// TIA Portal project "Tartak_Projekt" (V14)

(* hardware
DEVICE "S7-1200 station_1"  S7-1200 Station
   slot 0: "Rack_0"  S7-1200 Rack  Rack  V1.0
   slot 1: "PLC_1"  CPU 1214C DC/DC/DC  6ES7 214-1AG31-0XB0  V3.0
      slot 3: "AQ 1x12BIT_1"  AQ1 signal board  6ES7 232-4HA30-0XB0  V1.0
   slot 2: "DI 16/DQ 16x24VDC_1"  SM 1223 DI16/DQ16 x 24VDC  6ES7 223-1BL30-0XB0  V1.0
DEVICE "HMI_2"  TP700 Comfort
   slot 0: "TP700 Comfort"  TP700 Comfort  6AV2 124-0GC01-0AX0  14.0.1.0
   slot 1: "HMI_RT_2"  TP700 Comfort  6AV2 124-0GC01-0AX0  14.0.1.0
   slot 5: "HMI_1.IE_CP_1"  PROFINET Interface  14.0.1.0
      slot 1: "PROFINET Interface_1"  PROFINET Interface
         slot 1: "Port_1"  Port
         slot 2: "Port_2"  Port
   slot 7: "HMI_1.MPI/DP_CP_1"  MPI/DP Interface  14.0.1.0
*)

// ===== PLC "PLC_1"  CPU 1214C DC/DC/DC =====

VAR_GLOBAL   // PLC tag table "Non Default tag table2"
   "Tag_1" AT %M100.0 : Bool;
   "Tag_2" AT %M100.1 : Bool;
   "Tag_3" AT %M100.2 : Bool;
   "Tag_4" AT %M100.3 : Bool;
   "Tag_5" AT %M100.4 : Bool;
   "Tag_6" AT %M100.5 : Bool;
END_VAR

VAR_GLOBAL   // PLC tag table "Default tag table"
   "polozenie_dluga" AT %I8.0 : Bool;
   "polozenie_srednia" AT %I8.1 : Bool;
   "polozenie_krotka" AT %I8.2 : Bool;
   "polozenie_zsyp_krotki" AT %I8.3 : Bool;
   "polozenie_zsyp_sredni" AT %I8.4 : Bool;
   "polozenie_zsyp_dlugi" AT %I8.5 : Bool;
   "P1" AT %Q4.0 : Bool;   // Przepychacz belek krótkich
   "P2" AT %Q4.1 : Bool;   // Przepychacz belek średnich
   "P3" AT %Q4.2 : Bool;   // Przepychacz belek długich
   "otwarcie_zsyp_krotki" AT %Q4.3 : Bool;
   "otwarcie_zsyp_sredni" AT %Q4.4 : Bool;
   "otwarcie_zsyp_dlugi" AT %Q4.5 : Bool;
   "napelnienie_zsyp_krotki" AT %I8.6 : Bool;
   "napelnienie_zsyp_sredni" AT %I8.7 : Bool;
   "napelnienie_zsyp_dlugi" AT %I9.0 : Bool;
   "pozycja_wagnik_zsyp_krotki" AT %I9.7 : Bool;
   "pozycja_wagonik_zsyp_sredni" AT %I1.0 : Bool;
   "pozycja_wagonik_zsyp_dlugi" AT %I1.1 : Bool;
   "ruch_wagonika" AT %Q4.6 : Bool;
   "zwrotnica_bit_0" AT %Q4.7 : Bool;
   "zwrotnica_bit_1" AT %Q5.0 : Bool;
   "bocznica_krotka_0" AT %I9.1 : Bool;
   "bocznica_krotka_1" AT %I9.2 : Bool;
   "bocznica_srednia_0" AT %I9.3 : Bool;
   "bocznica_srednia_1" AT %I9.4 : Bool;
   "bocznica_dluga_0" AT %I9.5 : Bool;
   "bocznica_dluga_1" AT %I9.6 : Bool;
   "sygnalizator_dlugi" AT %Q5.1 : Bool;
   "sygnalizator_sredni" AT %Q5.2 : Bool;
   "sygnalizator_krotki" AT %Q5.3 : Bool;
   "Clock_Byte" AT %MB0 : Byte;
   "Clock_10Hz" AT %M0.0 : Bool;
   "Clock_5Hz" AT %M0.1 : Bool;
   "Clock_2.5Hz" AT %M0.2 : Bool;
   "Clock_2Hz" AT %M0.3 : Bool;
   "Clock_1.25Hz" AT %M0.4 : Bool;
   "Clock_1Hz" AT %M0.5 : Bool;
   "Clock_0.625Hz" AT %M0.6 : Bool;
   "Clock_0.5Hz" AT %M0.7 : Bool;
   "alarmy" AT %MW10 : Int;
END_VAR

VAR_GLOBAL CONSTANT   // PLC tag table "Default tag table"
   "None" : Pip := 65535;
   "Automatic update" : Pip := 0;
   "PIP 1" : Pip := 1;
   "PIP 2" : Pip := 2;
   "PIP 3" : Pip := 3;
   "PIP 4" : Pip := 4;
   "PIP OB Servo" : Pip := 32768;
   "Local~MC" : Hw_SubModule := 51;
   "Local~Common" : Hw_SubModule := 50;
   "Local~Device" : Hw_Device := 32;
   "Local~Configuration" : Hw_SubModule := 33;
   "Local~Exec" : Hw_SubModule := 52;
   "Local(1)" : Hw_SubModule := 49;
   "Local~PROFINET_interface_1(1)" : Hw_Interface := 64;
   "Local~PROFINET_interface_1~Port_1(1)" : Hw_Interface := 65;
   "Local~HSC_1(1)" : Hw_Hsc := 257;
   "Local~HSC_2(1)" : Hw_Hsc := 258;
   "Local~HSC_3(1)" : Hw_Hsc := 259;
   "Local~HSC_4(1)" : Hw_Hsc := 260;
   "Local~HSC_5(1)" : Hw_Hsc := 261;
   "Local~HSC_6(1)" : Hw_Hsc := 262;
   "Local~AI_2_1(1)" : Hw_SubModule := 263;
   "Local~DI_14_DQ_10_1(1)" : Hw_SubModule := 264;
   "Local~Pulse_1(1)" : Hw_Pwm := 265;
   "Local~Pulse_2(1)" : Hw_Pwm := 266;
   "Local~Pulse_3(1)" : Hw_Pwm := 267;
   "Local~Pulse_4(1)" : Hw_Pwm := 268;
   "OB_Main(1)" : OB_PCYCLE := 1;
END_VAR

DATA_BLOCK "DB_HMI"   // DB1
{ S7_Optimized_Access := 'TRUE' }
VERSION : 0.1
   VAR
      napelnienie_zsyp_krotki : Bool;
      napelnienie_zsyp_sredni : Bool;
      napelnienie_zsyp_dlugi : Bool;
      belka_krotka : Bool;
      belka_srednia : Bool;
      belka_dluga : Bool;
      status_ruchu_wagonika : Bool;
      oproznianie_zsyp_krotki : Bool;
      oproznianie_zsyp_sredni : Bool;
      oproznianie_zsyp_dlugi : Bool;
      ustawienie_zwrotnicy : Byte;
      zapelnienie_bocznicy_krotkiej : Byte;
      zapelnienie_bocznicy_sredniej : Byte;
      zapelnienie_bocznicy_dlugiej : Byte;
      sygnalizator_bocznica_krotka : Bool;
      sygnalizator_bocznica_srednia : Bool;
      sygnalizator_bocznica_dluga : Bool;
      wagonik_krotki : Bool;
      wagonik_sredni : Bool;
      wagonik_dlugi : Bool;
   END_VAR
BEGIN
END_DATA_BLOCK

DATA_BLOCK "wykrywanie_belki_i_zrzuczanie_DB"   // DB2
{ S7_Optimized_Access := 'TRUE' }
VERSION : 0.1
// stored: InstanceOfName wykrywanie_belki_i_zrzuczanie
"wykrywanie_belki_i_zrzuczanie"
BEGIN
END_DATA_BLOCK

DATA_BLOCK "poruszanie_wagonikiem_i_zsypywaanie_drewna_2_DB"   // DB3
{ S7_Optimized_Access := 'TRUE' }
VERSION : 0.1
// stored: InstanceOfName poruszanie_wagonikiem_i_zsypywaanie_drewna_2
"poruszanie_wagonikiem_i_zsypywaanie_drewna_2"
BEGIN
END_DATA_BLOCK

// folder: System blocks/Program resources

DATA_BLOCK "IEC_Timer_0_DB"   // DB4
{ S7_Optimized_Access := 'TRUE' }
AUTHOR : Simatic
FAMILY : IEC
NAME : IEC_TMR
VERSION : 1.0
// stored: InstanceOfName IEC_TIMER
"IEC_TIMER"
BEGIN
END_DATA_BLOCK

// folder: (top level)

FUNCTION_BLOCK "wykrywanie_belki_i_zrzuczanie"   // FB1, LAD
{ S7_Optimized_Access := 'TRUE' }
VERSION : 0.1
   VAR
      czy_wykryta_belka : Bool;
      krotka_belka : Bool;
      srednia_belka : Bool;
      dluga_belka : Bool;
      belka_zrzucona : Bool;
   END_VAR
   VAR_TEMP
      belka_na_pomiarze : Bool;
   END_VAR
   VAR_TEMP   // added for the SCL form of the ladder/FBD networks
      _w1 : Bool;
      _w2 : Bool;
      _w3 : Bool;
      _w4 : Bool;
   END_VAR
BEGIN

REGION Network 1
   // Czy belka jest już na pomiarze?
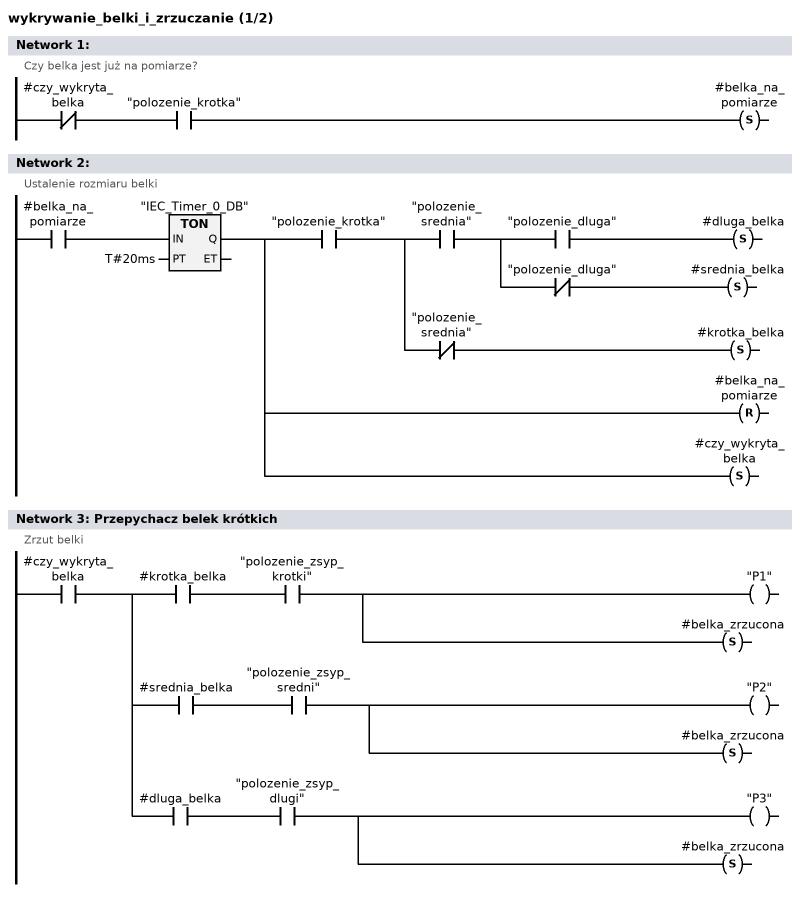
   RUNG wire#powerrail
      I_Contact( #czy_wykryta_belka )
      Contact( "polozenie_krotka" )
      S_Coil( #belka_na_pomiarze )
   END_RUNG
   // the same network as SCL:
   IF NOT #czy_wykryta_belka AND "polozenie_krotka" THEN #belka_na_pomiarze := TRUE; END_IF;
END_REGION

REGION Network 2
   // Ustalenie rozmiaru belki
   "IEC_Timer_0_DB".TON(IN := #belka_na_pomiarze, PT := T#20ms);
   #_w1 := "IEC_Timer_0_DB".Q AND "polozenie_krotka";
   #_w2 := #_w1 AND "polozenie_srednia";
   IF #_w2 AND "polozenie_dluga" THEN #dluga_belka := TRUE; END_IF;
   IF #_w2 AND NOT "polozenie_dluga" THEN #srednia_belka := TRUE; END_IF;
   IF #_w1 AND NOT "polozenie_srednia" THEN #krotka_belka := TRUE; END_IF;
   IF "IEC_Timer_0_DB".Q THEN
       #belka_na_pomiarze := FALSE;
       #czy_wykryta_belka := TRUE;
   END_IF;
END_REGION

REGION Network 3: Przepychacz belek krótkich
   // Zrzut belki
   RUNG wire#powerrail
      Contact( #czy_wykryta_belka )
      wire#w1
      Contact( #krotka_belka )
      Contact( "polozenie_zsyp_krotki" )
      wire#w2
      Coil( "P1" )
   END_RUNG
   RUNG wire#w2
      S_Coil( #belka_zrzucona )
   END_RUNG
   RUNG wire#w1
      Contact( #srednia_belka )
      Contact( "polozenie_zsyp_sredni" )
      wire#w3
      Coil( "P2" )
   END_RUNG
   RUNG wire#w3
      S_Coil( #belka_zrzucona )
   END_RUNG
   RUNG wire#w1
      Contact( #dluga_belka )
      Contact( "polozenie_zsyp_dlugi" )
      wire#w4
      Coil( "P3" )
   END_RUNG
   RUNG wire#w4
      S_Coil( #belka_zrzucona )
   END_RUNG
   // the same network as SCL:
   "P1" := #czy_wykryta_belka AND #krotka_belka AND "polozenie_zsyp_krotki";
   IF "P1" THEN #belka_zrzucona := TRUE; END_IF;
   "P2" := #czy_wykryta_belka AND #srednia_belka AND "polozenie_zsyp_sredni";
   IF "P2" THEN #belka_zrzucona := TRUE; END_IF;
   "P3" := #czy_wykryta_belka AND #dluga_belka AND "polozenie_zsyp_dlugi";
   IF "P3" THEN #belka_zrzucona := TRUE; END_IF;
END_REGION

REGION Network 4: Przepychacz belek krótkich
   // Czekamy, aż belka zostanie zrzucona
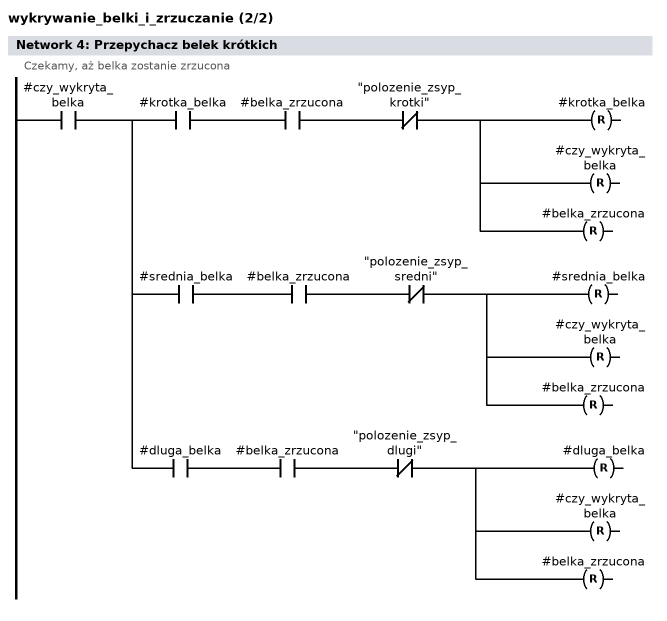
   RUNG wire#powerrail
      Contact( #czy_wykryta_belka )
      wire#w1
      Contact( #krotka_belka )
      Contact( #belka_zrzucona )
      I_Contact( "polozenie_zsyp_krotki" )
      wire#w2
      R_Coil( #krotka_belka )
   END_RUNG
   RUNG wire#w2
      R_Coil( #czy_wykryta_belka )
   END_RUNG
   RUNG wire#w2
      R_Coil( #belka_zrzucona )
   END_RUNG
   RUNG wire#w1
      Contact( #srednia_belka )
      Contact( #belka_zrzucona )
      I_Contact( "polozenie_zsyp_sredni" )
      wire#w3
      R_Coil( #srednia_belka )
   END_RUNG
   RUNG wire#w3
      R_Coil( #czy_wykryta_belka )
   END_RUNG
   RUNG wire#w3
      R_Coil( #belka_zrzucona )
   END_RUNG
   RUNG wire#w1
      Contact( #dluga_belka )
      Contact( #belka_zrzucona )
      I_Contact( "polozenie_zsyp_dlugi" )
      wire#w4
      R_Coil( #dluga_belka )
   END_RUNG
   RUNG wire#w4
      R_Coil( #czy_wykryta_belka )
   END_RUNG
   RUNG wire#w4
      R_Coil( #belka_zrzucona )
   END_RUNG
   // the same network as SCL:
   #_w1 := #czy_wykryta_belka AND #krotka_belka AND #belka_zrzucona AND NOT "polozenie_zsyp_krotki";
   IF #_w1 THEN #krotka_belka := FALSE; END_IF;
   #_w2 := #czy_wykryta_belka;
   IF #_w1 THEN
       #czy_wykryta_belka := FALSE;
       #belka_zrzucona := FALSE;
   END_IF;
   #_w3 := #_w2 AND #srednia_belka AND #belka_zrzucona AND NOT "polozenie_zsyp_sredni";
   IF #_w3 THEN
       #srednia_belka := FALSE;
       #czy_wykryta_belka := FALSE;
       #belka_zrzucona := FALSE;
   END_IF;
   #_w4 := #_w2 AND #dluga_belka AND #belka_zrzucona AND NOT "polozenie_zsyp_dlugi";
   IF #_w4 THEN
       #dluga_belka := FALSE;
       #czy_wykryta_belka := FALSE;
       #belka_zrzucona := FALSE;
   END_IF;
END_REGION
END_FUNCTION_BLOCK

FUNCTION_BLOCK "poruszanie_wagonikiem_i_zsypywaanie_drewna_2"   // FB2, LAD
{ S7_Optimized_Access := 'TRUE' }
VERSION : 0.1
   VAR
      wagonik_krotki : Bool;
      wagonik_sredni : Bool;
      wagonik_dlugi : Bool;
   END_VAR
   VAR_TEMP   // added for the SCL form of the ladder/FBD networks
      _w1 : Bool;
      _w2 : Bool;
      _w3 : Bool;
      _w4 : Bool;
      _w5 : Bool;
      _w6 : Bool;
   END_VAR
BEGIN

REGION Network 1
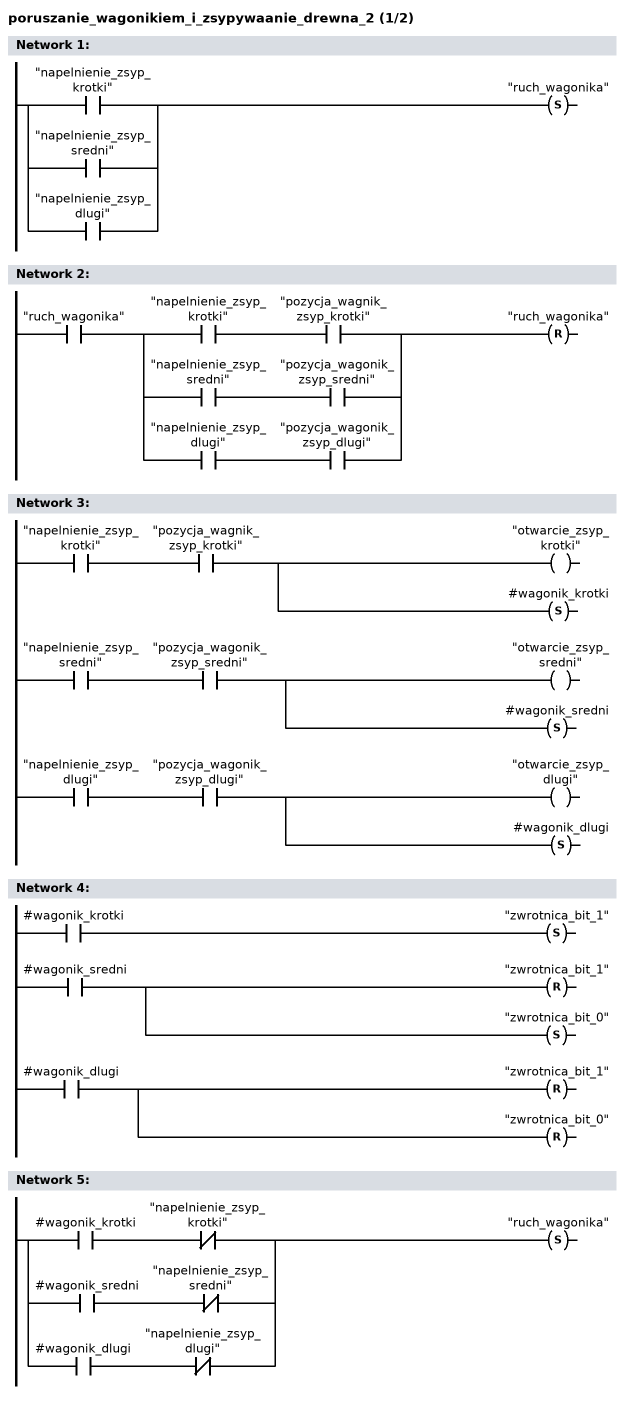
   RUNG wire#powerrail
      Contact( "napelnienie_zsyp_krotki" )
      wire#w1
      S_Coil( "ruch_wagonika" )
   END_RUNG
   RUNG wire#powerrail
      Contact( "napelnienie_zsyp_sredni" )
   END_RUNG wire#w1
   RUNG wire#powerrail
      Contact( "napelnienie_zsyp_dlugi" )
   END_RUNG wire#w1
   // the same network as SCL:
   IF "napelnienie_zsyp_krotki" OR "napelnienie_zsyp_sredni" OR "napelnienie_zsyp_dlugi" THEN
       "ruch_wagonika" := TRUE;
   END_IF;
END_REGION

REGION Network 2
   RUNG wire#powerrail
      Contact( "ruch_wagonika" )
      wire#w1
      Contact( "napelnienie_zsyp_krotki" )
      Contact( "pozycja_wagnik_zsyp_krotki" )
      wire#w2
      R_Coil( "ruch_wagonika" )
   END_RUNG
   RUNG wire#w1
      Contact( "napelnienie_zsyp_sredni" )
      Contact( "pozycja_wagonik_zsyp_sredni" )
   END_RUNG wire#w2
   RUNG wire#w1
      Contact( "napelnienie_zsyp_dlugi" )
      Contact( "pozycja_wagonik_zsyp_dlugi" )
   END_RUNG wire#w2
   // the same network as SCL:
   IF "ruch_wagonika" AND (("napelnienie_zsyp_krotki" AND "pozycja_wagnik_zsyp_krotki") OR ("napelnienie_zsyp_sredni" AND "pozycja_wagonik_zsyp_sredni") OR ("napelnienie_zsyp_dlugi" AND "pozycja_wagonik_zsyp_dlugi")) THEN
       "ruch_wagonika" := FALSE;
   END_IF;
END_REGION

REGION Network 3
   RUNG wire#powerrail
      Contact( "napelnienie_zsyp_krotki" )
      Contact( "pozycja_wagnik_zsyp_krotki" )
      wire#w1
      Coil( "otwarcie_zsyp_krotki" )
   END_RUNG
   RUNG wire#w1
      S_Coil( #wagonik_krotki )
   END_RUNG
   RUNG wire#powerrail
      Contact( "napelnienie_zsyp_sredni" )
      Contact( "pozycja_wagonik_zsyp_sredni" )
      wire#w2
      Coil( "otwarcie_zsyp_sredni" )
   END_RUNG
   RUNG wire#w2
      S_Coil( #wagonik_sredni )
   END_RUNG
   RUNG wire#powerrail
      Contact( "napelnienie_zsyp_dlugi" )
      Contact( "pozycja_wagonik_zsyp_dlugi" )
      wire#w3
      Coil( "otwarcie_zsyp_dlugi" )
   END_RUNG
   RUNG wire#w3
      S_Coil( #wagonik_dlugi )
   END_RUNG
   // the same network as SCL:
   "otwarcie_zsyp_krotki" := "napelnienie_zsyp_krotki" AND "pozycja_wagnik_zsyp_krotki";
   IF "otwarcie_zsyp_krotki" THEN #wagonik_krotki := TRUE; END_IF;
   "otwarcie_zsyp_sredni" := "napelnienie_zsyp_sredni" AND "pozycja_wagonik_zsyp_sredni";
   IF "otwarcie_zsyp_sredni" THEN #wagonik_sredni := TRUE; END_IF;
   "otwarcie_zsyp_dlugi" := "napelnienie_zsyp_dlugi" AND "pozycja_wagonik_zsyp_dlugi";
   IF "otwarcie_zsyp_dlugi" THEN #wagonik_dlugi := TRUE; END_IF;
END_REGION

REGION Network 4
   RUNG wire#powerrail
      Contact( #wagonik_krotki )
      S_Coil( "zwrotnica_bit_1" )
   END_RUNG
   RUNG wire#powerrail
      Contact( #wagonik_sredni )
      wire#w1
      R_Coil( "zwrotnica_bit_1" )
   END_RUNG
   RUNG wire#w1
      S_Coil( "zwrotnica_bit_0" )
   END_RUNG
   RUNG wire#powerrail
      Contact( #wagonik_dlugi )
      wire#w2
      R_Coil( "zwrotnica_bit_1" )
   END_RUNG
   RUNG wire#w2
      R_Coil( "zwrotnica_bit_0" )
   END_RUNG
   // the same network as SCL:
   IF #wagonik_krotki THEN "zwrotnica_bit_1" := TRUE; END_IF;
   IF #wagonik_sredni THEN
       "zwrotnica_bit_1" := FALSE;
       "zwrotnica_bit_0" := TRUE;
   END_IF;
   IF #wagonik_dlugi THEN
       "zwrotnica_bit_1" := FALSE;
       "zwrotnica_bit_0" := FALSE;
   END_IF;
END_REGION

REGION Network 5
   RUNG wire#powerrail
      Contact( #wagonik_krotki )
      I_Contact( "napelnienie_zsyp_krotki" )
      wire#w1
      S_Coil( "ruch_wagonika" )
   END_RUNG
   RUNG wire#powerrail
      Contact( #wagonik_sredni )
      I_Contact( "napelnienie_zsyp_sredni" )
   END_RUNG wire#w1
   RUNG wire#powerrail
      Contact( #wagonik_dlugi )
      I_Contact( "napelnienie_zsyp_dlugi" )
   END_RUNG wire#w1
   // the same network as SCL:
   IF (#wagonik_krotki AND NOT "napelnienie_zsyp_krotki") OR (#wagonik_sredni AND NOT "napelnienie_zsyp_sredni") OR (#wagonik_dlugi AND NOT "napelnienie_zsyp_dlugi") THEN
       "ruch_wagonika" := TRUE;
   END_IF;
END_REGION

REGION Network 6
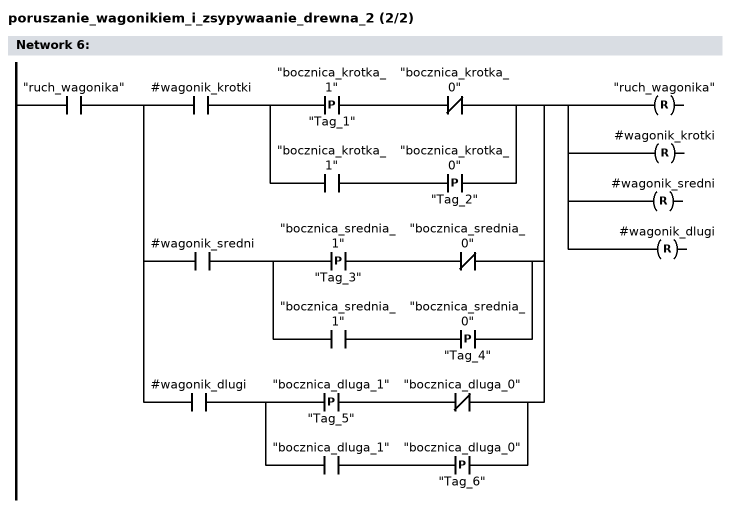
   RUNG wire#powerrail
      Contact( "ruch_wagonika" )
      wire#w1
      Contact( #wagonik_krotki )
      wire#w2
      P_Contact(operand := "bocznica_krotka_1", bit := "Tag_1")
      I_Contact( "bocznica_krotka_0" )
      wire#w3
      R_Coil( "ruch_wagonika" )
   END_RUNG
   RUNG wire#w2
      Contact( "bocznica_krotka_1" )
      P_Contact(operand := "bocznica_krotka_0", bit := "Tag_2")
   END_RUNG wire#w3
   RUNG wire#w1
      Contact( #wagonik_sredni )
      wire#w4
      P_Contact(operand := "bocznica_srednia_1", bit := "Tag_3")
      I_Contact( "bocznica_srednia_0" )
   END_RUNG wire#w3
   RUNG wire#w4
      Contact( "bocznica_srednia_1" )
      P_Contact(operand := "bocznica_srednia_0", bit := "Tag_4")
   END_RUNG wire#w3
   RUNG wire#w1
      Contact( #wagonik_dlugi )
      wire#w5
      P_Contact(operand := "bocznica_dluga_1", bit := "Tag_5")
      I_Contact( "bocznica_dluga_0" )
   END_RUNG wire#w3
   RUNG wire#w5
      Contact( "bocznica_dluga_1" )
      P_Contact(operand := "bocznica_dluga_0", bit := "Tag_6")
   END_RUNG wire#w3
   RUNG wire#w3
      R_Coil( #wagonik_krotki )
   END_RUNG
   RUNG wire#w3
      R_Coil( #wagonik_sredni )
   END_RUNG
   RUNG wire#w3
      R_Coil( #wagonik_dlugi )
   END_RUNG
   // the same network as SCL:
   #_w1 := "ruch_wagonika" AND #wagonik_krotki AND "bocznica_krotka_1" AND NOT "Tag_1";   // rising edge of "bocznica_krotka_1"
   "Tag_1" := "bocznica_krotka_1";
   #_w2 := "ruch_wagonika" AND #wagonik_krotki AND "bocznica_krotka_1" AND "bocznica_krotka_0" AND NOT "Tag_2";   // rising edge of "bocznica_krotka_0"
   "Tag_2" := "bocznica_krotka_0";
   #_w3 := "ruch_wagonika" AND #wagonik_sredni AND "bocznica_srednia_1" AND NOT "Tag_3";   // rising edge of "bocznica_srednia_1"
   "Tag_3" := "bocznica_srednia_1";
   #_w4 := "ruch_wagonika" AND #wagonik_sredni AND "bocznica_srednia_1" AND "bocznica_srednia_0" AND NOT "Tag_4";   // rising edge of "bocznica_srednia_0"
   "Tag_4" := "bocznica_srednia_0";
   #_w5 := "ruch_wagonika" AND #wagonik_dlugi AND "bocznica_dluga_1" AND NOT "Tag_5";   // rising edge of "bocznica_dluga_1"
   "Tag_5" := "bocznica_dluga_1";
   #_w6 := "ruch_wagonika" AND #wagonik_dlugi AND "bocznica_dluga_1" AND "bocznica_dluga_0" AND NOT "Tag_6";   // rising edge of "bocznica_dluga_0"
   "Tag_6" := "bocznica_dluga_0";
   IF (#_w1 AND NOT "bocznica_krotka_0") OR #_w2 OR (#_w3 AND NOT "bocznica_srednia_0") OR #_w4 OR (#_w5 AND NOT "bocznica_dluga_0") OR #_w6 THEN
       "ruch_wagonika" := FALSE;
       #wagonik_krotki := FALSE;
       #wagonik_sredni := FALSE;
       #wagonik_dlugi := FALSE;
   END_IF;
END_REGION
END_FUNCTION_BLOCK

FUNCTION "przepisywanie_HMI" : Void   // FC1, LAD
{ S7_Optimized_Access := 'TRUE' }
VERSION : 0.1
BEGIN

REGION Network 1: Napełnianie zsypów
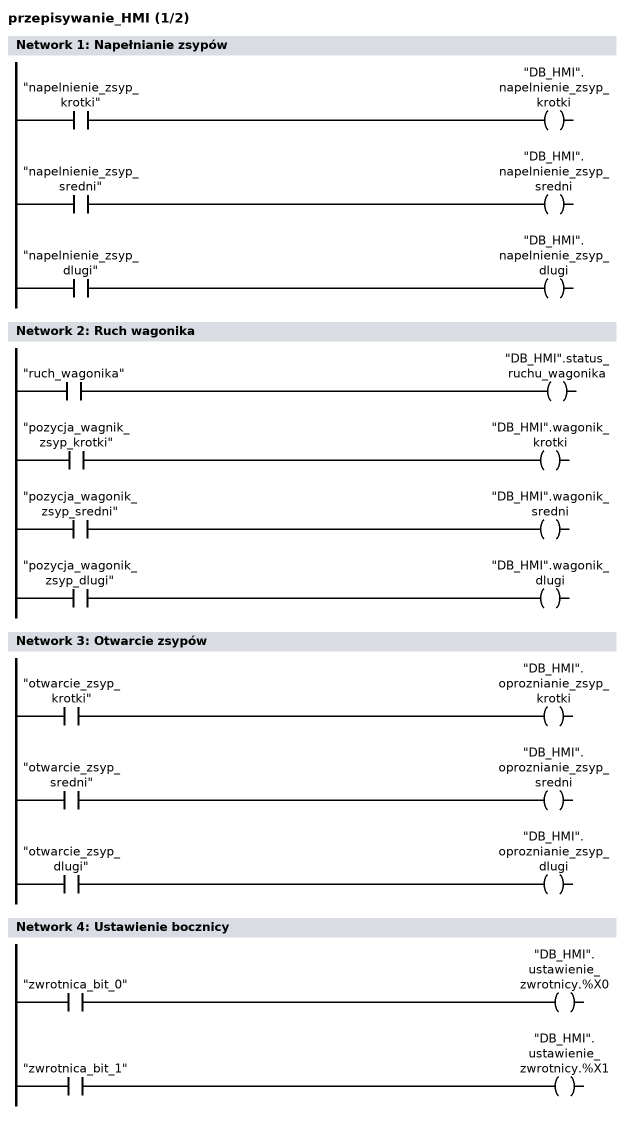
   RUNG wire#powerrail
      Contact( "napelnienie_zsyp_krotki" )
      Coil( "DB_HMI".napelnienie_zsyp_krotki )
   END_RUNG
   RUNG wire#powerrail
      Contact( "napelnienie_zsyp_sredni" )
      Coil( "DB_HMI".napelnienie_zsyp_sredni )
   END_RUNG
   RUNG wire#powerrail
      Contact( "napelnienie_zsyp_dlugi" )
      Coil( "DB_HMI".napelnienie_zsyp_dlugi )
   END_RUNG
   // the same network as SCL:
   "DB_HMI".napelnienie_zsyp_krotki := "napelnienie_zsyp_krotki";
   "DB_HMI".napelnienie_zsyp_sredni := "napelnienie_zsyp_sredni";
   "DB_HMI".napelnienie_zsyp_dlugi := "napelnienie_zsyp_dlugi";
END_REGION

REGION Network 2: Ruch wagonika
   RUNG wire#powerrail
      Contact( "ruch_wagonika" )
      Coil( "DB_HMI".status_ruchu_wagonika )
   END_RUNG
   RUNG wire#powerrail
      Contact( "pozycja_wagnik_zsyp_krotki" )
      Coil( "DB_HMI".wagonik_krotki )
   END_RUNG
   RUNG wire#powerrail
      Contact( "pozycja_wagonik_zsyp_sredni" )
      Coil( "DB_HMI".wagonik_sredni )
   END_RUNG
   RUNG wire#powerrail
      Contact( "pozycja_wagonik_zsyp_dlugi" )
      Coil( "DB_HMI".wagonik_dlugi )
   END_RUNG
   // the same network as SCL:
   "DB_HMI".status_ruchu_wagonika := "ruch_wagonika";
   "DB_HMI".wagonik_krotki := "pozycja_wagnik_zsyp_krotki";
   "DB_HMI".wagonik_sredni := "pozycja_wagonik_zsyp_sredni";
   "DB_HMI".wagonik_dlugi := "pozycja_wagonik_zsyp_dlugi";
END_REGION

REGION Network 3: Otwarcie zsypów
   RUNG wire#powerrail
      Contact( "otwarcie_zsyp_krotki" )
      Coil( "DB_HMI".oproznianie_zsyp_krotki )
   END_RUNG
   RUNG wire#powerrail
      Contact( "otwarcie_zsyp_sredni" )
      Coil( "DB_HMI".oproznianie_zsyp_sredni )
   END_RUNG
   RUNG wire#powerrail
      Contact( "otwarcie_zsyp_dlugi" )
      Coil( "DB_HMI".oproznianie_zsyp_dlugi )
   END_RUNG
   // the same network as SCL:
   "DB_HMI".oproznianie_zsyp_krotki := "otwarcie_zsyp_krotki";
   "DB_HMI".oproznianie_zsyp_sredni := "otwarcie_zsyp_sredni";
   "DB_HMI".oproznianie_zsyp_dlugi := "otwarcie_zsyp_dlugi";
END_REGION

REGION Network 4: Ustawienie bocznicy
   RUNG wire#powerrail
      Contact( "zwrotnica_bit_0" )
      Coil( "DB_HMI".ustawienie_zwrotnicy.%X0 )
   END_RUNG
   RUNG wire#powerrail
      Contact( "zwrotnica_bit_1" )
      Coil( "DB_HMI".ustawienie_zwrotnicy.%X1 )
   END_RUNG
   // the same network as SCL:
   "DB_HMI".ustawienie_zwrotnicy.%X0 := "zwrotnica_bit_0";
   "DB_HMI".ustawienie_zwrotnicy.%X1 := "zwrotnica_bit_1";
END_REGION

REGION Network 5: Zapełnienie bocznic
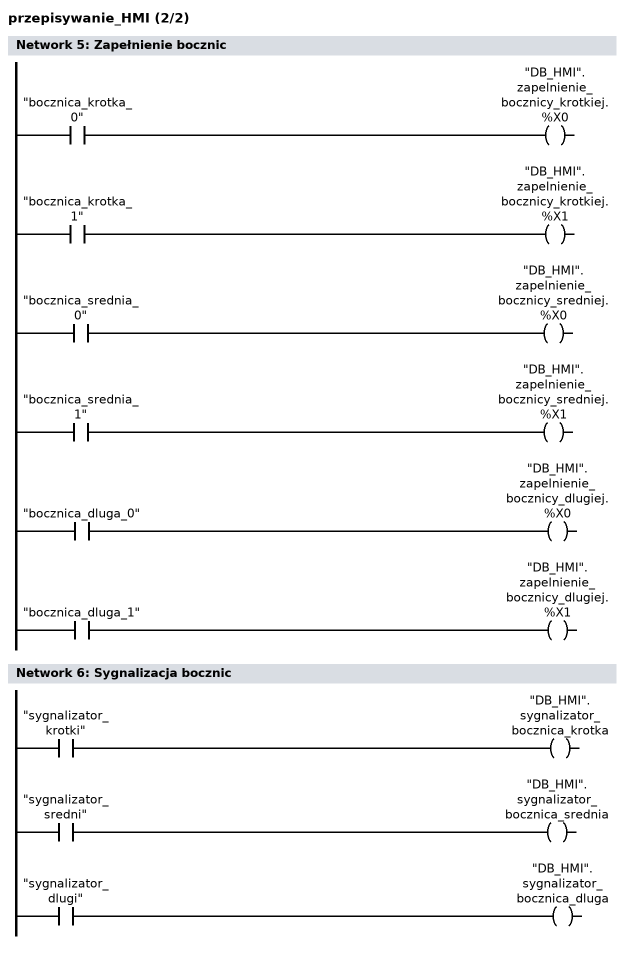
   RUNG wire#powerrail
      Contact( "bocznica_krotka_0" )
      Coil( "DB_HMI".zapelnienie_bocznicy_krotkiej.%X0 )
   END_RUNG
   RUNG wire#powerrail
      Contact( "bocznica_krotka_1" )
      Coil( "DB_HMI".zapelnienie_bocznicy_krotkiej.%X1 )
   END_RUNG
   RUNG wire#powerrail
      Contact( "bocznica_srednia_0" )
      Coil( "DB_HMI".zapelnienie_bocznicy_sredniej.%X0 )
   END_RUNG
   RUNG wire#powerrail
      Contact( "bocznica_srednia_1" )
      Coil( "DB_HMI".zapelnienie_bocznicy_sredniej.%X1 )
   END_RUNG
   RUNG wire#powerrail
      Contact( "bocznica_dluga_0" )
      Coil( "DB_HMI".zapelnienie_bocznicy_dlugiej.%X0 )
   END_RUNG
   RUNG wire#powerrail
      Contact( "bocznica_dluga_1" )
      Coil( "DB_HMI".zapelnienie_bocznicy_dlugiej.%X1 )
   END_RUNG
   // the same network as SCL:
   "DB_HMI".zapelnienie_bocznicy_krotkiej.%X0 := "bocznica_krotka_0";
   "DB_HMI".zapelnienie_bocznicy_krotkiej.%X1 := "bocznica_krotka_1";
   "DB_HMI".zapelnienie_bocznicy_sredniej.%X0 := "bocznica_srednia_0";
   "DB_HMI".zapelnienie_bocznicy_sredniej.%X1 := "bocznica_srednia_1";
   "DB_HMI".zapelnienie_bocznicy_dlugiej.%X0 := "bocznica_dluga_0";
   "DB_HMI".zapelnienie_bocznicy_dlugiej.%X1 := "bocznica_dluga_1";
END_REGION

REGION Network 6: Sygnalizacja bocznic
   RUNG wire#powerrail
      Contact( "sygnalizator_krotki" )
      Coil( "DB_HMI".sygnalizator_bocznica_krotka )
   END_RUNG
   RUNG wire#powerrail
      Contact( "sygnalizator_sredni" )
      Coil( "DB_HMI".sygnalizator_bocznica_srednia )
   END_RUNG
   RUNG wire#powerrail
      Contact( "sygnalizator_dlugi" )
      Coil( "DB_HMI".sygnalizator_bocznica_dluga )
   END_RUNG
   // the same network as SCL:
   "DB_HMI".sygnalizator_bocznica_krotka := "sygnalizator_krotki";
   "DB_HMI".sygnalizator_bocznica_srednia := "sygnalizator_sredni";
   "DB_HMI".sygnalizator_bocznica_dluga := "sygnalizator_dlugi";
END_REGION
END_FUNCTION

FUNCTION "poruszanie_wagonikiem_i_zsypywanie_drewna" : Void   // FC2, LAD
{ S7_Optimized_Access := 'TRUE' }
VERSION : 0.1
BEGIN

REGION Network 1
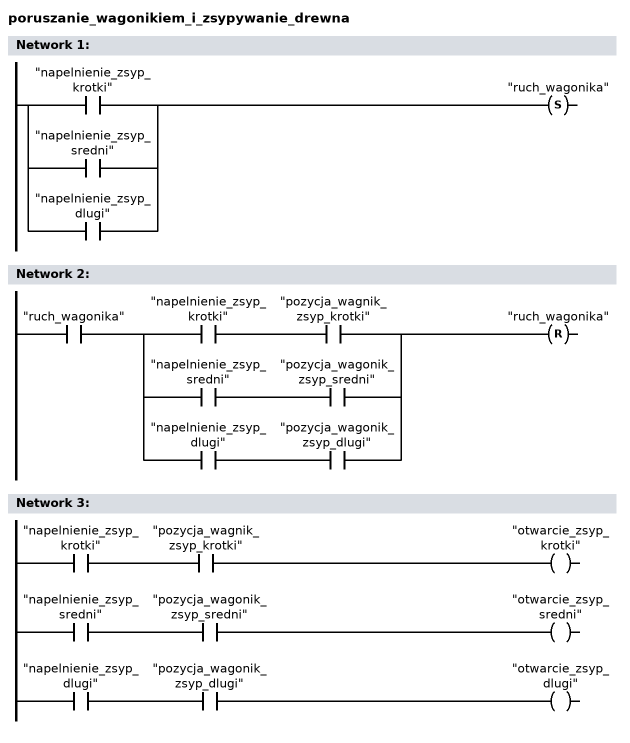
   RUNG wire#powerrail
      Contact( "napelnienie_zsyp_krotki" )
      wire#w1
      S_Coil( "ruch_wagonika" )
   END_RUNG
   RUNG wire#powerrail
      Contact( "napelnienie_zsyp_sredni" )
   END_RUNG wire#w1
   RUNG wire#powerrail
      Contact( "napelnienie_zsyp_dlugi" )
   END_RUNG wire#w1
   // the same network as SCL:
   IF "napelnienie_zsyp_krotki" OR "napelnienie_zsyp_sredni" OR "napelnienie_zsyp_dlugi" THEN
       "ruch_wagonika" := TRUE;
   END_IF;
END_REGION

REGION Network 2
   RUNG wire#powerrail
      Contact( "ruch_wagonika" )
      wire#w1
      Contact( "napelnienie_zsyp_krotki" )
      Contact( "pozycja_wagnik_zsyp_krotki" )
      wire#w2
      R_Coil( "ruch_wagonika" )
   END_RUNG
   RUNG wire#w1
      Contact( "napelnienie_zsyp_sredni" )
      Contact( "pozycja_wagonik_zsyp_sredni" )
   END_RUNG wire#w2
   RUNG wire#w1
      Contact( "napelnienie_zsyp_dlugi" )
      Contact( "pozycja_wagonik_zsyp_dlugi" )
   END_RUNG wire#w2
   // the same network as SCL:
   IF "ruch_wagonika" AND (("napelnienie_zsyp_krotki" AND "pozycja_wagnik_zsyp_krotki") OR ("napelnienie_zsyp_sredni" AND "pozycja_wagonik_zsyp_sredni") OR ("napelnienie_zsyp_dlugi" AND "pozycja_wagonik_zsyp_dlugi")) THEN
       "ruch_wagonika" := FALSE;
   END_IF;
END_REGION

REGION Network 3
   RUNG wire#powerrail
      Contact( "napelnienie_zsyp_krotki" )
      Contact( "pozycja_wagnik_zsyp_krotki" )
      Coil( "otwarcie_zsyp_krotki" )
   END_RUNG
   RUNG wire#powerrail
      Contact( "napelnienie_zsyp_sredni" )
      Contact( "pozycja_wagonik_zsyp_sredni" )
      Coil( "otwarcie_zsyp_sredni" )
   END_RUNG
   RUNG wire#powerrail
      Contact( "napelnienie_zsyp_dlugi" )
      Contact( "pozycja_wagonik_zsyp_dlugi" )
      Coil( "otwarcie_zsyp_dlugi" )
   END_RUNG
   // the same network as SCL:
   "otwarcie_zsyp_krotki" := "napelnienie_zsyp_krotki" AND "pozycja_wagnik_zsyp_krotki";
   "otwarcie_zsyp_sredni" := "napelnienie_zsyp_sredni" AND "pozycja_wagonik_zsyp_sredni";
   "otwarcie_zsyp_dlugi" := "napelnienie_zsyp_dlugi" AND "pozycja_wagonik_zsyp_dlugi";
END_REGION
END_FUNCTION

FUNCTION "opuszczanie_tartaku" : Void   // FC3, LAD
{ S7_Optimized_Access := 'TRUE' }
VERSION : 0.1
BEGIN

REGION Network 1
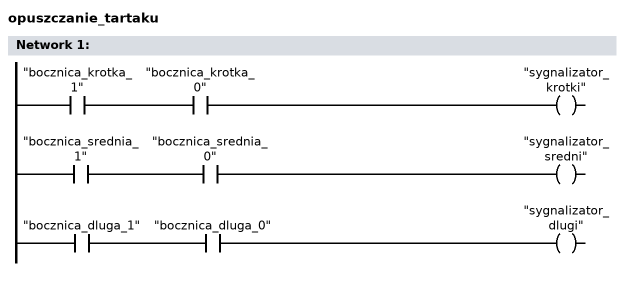
   RUNG wire#powerrail
      Contact( "bocznica_krotka_1" )
      Contact( "bocznica_krotka_0" )
      Coil( "sygnalizator_krotki" )
   END_RUNG
   RUNG wire#powerrail
      Contact( "bocznica_srednia_1" )
      Contact( "bocznica_srednia_0" )
      Coil( "sygnalizator_sredni" )
   END_RUNG
   RUNG wire#powerrail
      Contact( "bocznica_dluga_1" )
      Contact( "bocznica_dluga_0" )
      Coil( "sygnalizator_dlugi" )
   END_RUNG
   // the same network as SCL:
   "sygnalizator_krotki" := "bocznica_krotka_1" AND "bocznica_krotka_0";
   "sygnalizator_sredni" := "bocznica_srednia_1" AND "bocznica_srednia_0";
   "sygnalizator_dlugi" := "bocznica_dluga_1" AND "bocznica_dluga_0";
END_REGION
END_FUNCTION

ORGANIZATION_BLOCK "Main"   // OB1, LAD, ProgramCycle
TITLE = "Main Program Sweep (Cycle)"
{ S7_Optimized_Access := 'TRUE' }
VERSION : 0.1
   VAR_INPUT
      Initial_Call : Bool;   // Initial call of this OB
      Remanence : Bool;   // =True, if remanent data are available
   END_VAR
BEGIN

REGION Network 1
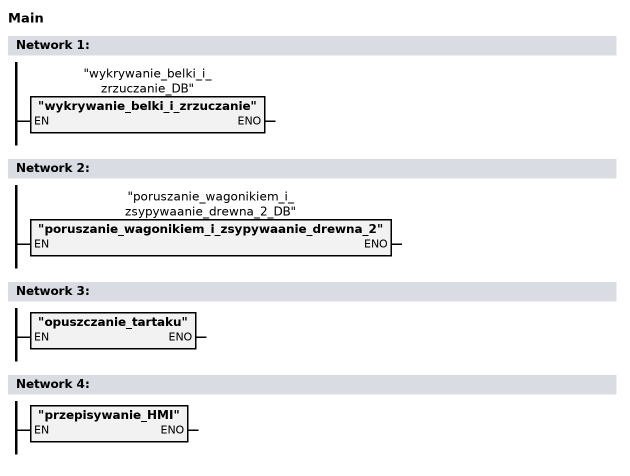
   RUNG wire#powerrail
      "wykrywanie_belki_i_zrzuczanie_DB"()
   END_RUNG
   // the same network as SCL:
   "wykrywanie_belki_i_zrzuczanie_DB"();   // "wykrywanie_belki_i_zrzuczanie"
END_REGION

REGION Network 2
   RUNG wire#powerrail
      "poruszanie_wagonikiem_i_zsypywaanie_drewna_2_DB"()
   END_RUNG
   // the same network as SCL:
   "poruszanie_wagonikiem_i_zsypywaanie_drewna_2_DB"();   // "poruszanie_wagonikiem_i_zsypywaanie_drewna_2"
END_REGION

REGION Network 3
   RUNG wire#powerrail
      "opuszczanie_tartaku"()
   END_RUNG
   // the same network as SCL:
   "opuszczanie_tartaku"();
END_REGION

REGION Network 4
   RUNG wire#powerrail
      "przepisywanie_HMI"()
   END_RUNG
   // the same network as SCL:
   "przepisywanie_HMI"();
END_REGION
END_ORGANIZATION_BLOCK

(* ===== HMI "HMI_RT_2" =====
system functions are stored by id; their names below are inferred from use
connection "HMI_Connection_1": ETHERNET, S7_1200_OMS

HMI tags "Default tag table"
   "Tag_ScreenNumber" : UInt, internal
   "DB_HMI_napelnienie_zsyp_krotki" : Bool = PLC DB_HMI.napelnienie_zsyp_krotki, 1 s
   "DB_HMI_napelnienie_zsyp_sredni" : Bool = PLC DB_HMI.napelnienie_zsyp_sredni, 1 s
   "DB_HMI_napelnienie_zsyp_dlugi" : Bool = PLC DB_HMI.napelnienie_zsyp_dlugi, 1 s
   "DB_HMI_oproznianie_zsyp_krotki" : Bool = PLC DB_HMI.oproznianie_zsyp_krotki, 1 s
   "DB_HMI_oproznianie_zsyp_sredni" : Bool = PLC DB_HMI.oproznianie_zsyp_sredni, 1 s
   "DB_HMI_oproznianie_zsyp_dlugi" : Bool = PLC DB_HMI.oproznianie_zsyp_dlugi, 1 s
   "DB_HMI_status_ruchu_wagonika" : Bool = PLC DB_HMI.status_ruchu_wagonika, 1 s
   "DB_HMI_wagonik_dlugi" : Bool = PLC DB_HMI.wagonik_dlugi, 1 s
   "DB_HMI_wagonik_sredni" : Bool = PLC DB_HMI.wagonik_sredni, 1 s
   "DB_HMI_wagonik_krotki" : Bool = PLC DB_HMI.wagonik_krotki, 1 s
   "DB_HMI_zapelnienie_bocznicy_dlugiej" : Byte = PLC DB_HMI.zapelnienie_bocznicy_dlugiej, 1 s
   "DB_HMI_sygnalizator_bocznica_srednia" : Bool = PLC DB_HMI.sygnalizator_bocznica_srednia, 1 s
   "DB_HMI_zapelnienie_bocznicy_sredniej" : Byte = PLC DB_HMI.zapelnienie_bocznicy_sredniej, 1 s
   "DB_HMI_zapelnienie_bocznicy_krotkiej" : Byte = PLC DB_HMI.zapelnienie_bocznicy_krotkiej, 1 s
   "DB_HMI_sygnalizator_bocznica_dluga" : Bool = PLC DB_HMI.sygnalizator_bocznica_dluga, 1 s
   "DB_HMI_sygnalizator_bocznica_krotka" : Bool = PLC DB_HMI.sygnalizator_bocznica_krotka, 1 s
   "DB_HMI_ustawienie_zwrotnicy" : Byte = PLC DB_HMI.ustawienie_zwrotnicy, 1 s

screen "Root screen" 800x420, template "Template_1"
   on GenerateScreen: SetTag("Tag_ScreenNumber", 1)
   SymbolLibrary "Symbol library_3" at 594,75 size 73x103
      Appearance <- "DB_HMI_napelnienie_zsyp_dlugi"
   SymbolLibrary "Symbol library_2" at 487,75 size 73x103
      Appearance <- "DB_HMI_napelnienie_zsyp_sredni"
   SymbolLibrary "Symbol library_1" at 380,75 size 73x103
      Appearance <- "DB_HMI_napelnienie_zsyp_krotki"
   GraphicIOField "PlotLight_Round_G" at 405,148 size 22x21; PictureOff "PilotLight_Round_G_Off_256c"; PictureOn "PilotLight_Round_G_On_256c"
      ProcessValue <- "DB_HMI_oproznianie_zsyp_krotki"
   GraphicIOField "PlotLight_Round_G_1" at 512,150 size 22x21; PictureOn "PilotLight_Round_G_On_256c"; PictureOff "PilotLight_Round_G_Off_256c"
      ProcessValue <- "DB_HMI_oproznianie_zsyp_sredni"
   GraphicIOField "PlotLight_Round_G_2" at 619,149 size 22x21; PictureOff "PilotLight_Round_G_Off_256c"; PictureOn "PilotLight_Round_G_On_256c"
      ProcessValue <- "DB_HMI_napelnienie_zsyp_dlugi"
   GraphicIOField "PlotLight_Square_G" at 731,262 size 50x50; PictureOff "PilotLight_Square_G_Off_256c"; PictureOn "PilotLight_Square_G_On_256c"
      ProcessValue <- "DB_HMI_status_ruchu_wagonika"
   GraphicView "Graphic view_4" at 596,194 size 80x74; Picture "Graphic_5"
      Visibility <- "DB_HMI_wagonik_dlugi"
   GraphicView "Graphic view_5" at 487,194 size 80x74; Picture "Graphic_5"
      Visibility <- "DB_HMI_wagonik_sredni"
   GraphicView "Graphic view_6" at 376,194 size 80x74; Picture "Graphic_5"
      Visibility <- "DB_HMI_wagonik_krotki"
   GraphicView "Graphic view_7" at 48,133 size 63x62; Picture "Graphic_5"
      Visibility <- "DB_HMI_zapelnienie_bocznicy_dlugiej"
   GraphicView "Graphic view_8" at 124,133 size 63x62; Picture "Graphic_5"
      Visibility <- "DB_HMI_zapelnienie_bocznicy_dlugiej"
   GraphicView "Graphic view_9" at 49,207 size 63x62; Picture "Graphic_5"
      Visibility <- "DB_HMI_zapelnienie_bocznicy_sredniej"
   GraphicView "Graphic view_10" at 125,207 size 63x62; Picture "Graphic_5"
      Visibility <- "DB_HMI_zapelnienie_bocznicy_sredniej"
   GraphicView "Graphic view_11" at 48,285 size 63x62; Picture "Graphic_5"
      Visibility <- "DB_HMI_zapelnienie_bocznicy_krotkiej"
   GraphicView "Graphic view_12" at 124,285 size 63x62; Picture "Graphic_5"
      Visibility <- "DB_HMI_zapelnienie_bocznicy_krotkiej"
   Line "Line_5" at 199,196 size 84x76
      Visibility <- "DB_HMI_ustawienie_zwrotnicy"
   Line "Line_6" at 200,272 size 82x0
      Visibility <- "DB_HMI_ustawienie_zwrotnicy"
   Line "Line_7" at 198,273 size 84x77
      Visibility <- "DB_HMI_ustawienie_zwrotnicy"
   GraphicIOField "PlotLight_Round_G_3" at 14,132 size 28x27; PictureOff "PilotLight_Round_G_Off_256c"; PictureOn "PilotLight_Round_G_On_256c"
      ProcessValue <- "DB_HMI_sygnalizator_bocznica_dluga"
   GraphicIOField "PlotLight_Round_G_4" at 12,206 size 28x27; PictureOn "PilotLight_Round_G_On_256c"; PictureOff "PilotLight_Round_G_Off_256c"
      ProcessValue <- "DB_HMI_sygnalizator_bocznica_srednia"
   GraphicIOField "PlotLight_Round_G_5" at 12,284 size 28x27; PictureOff "PilotLight_Round_G_Off_256c"; PictureOn "PilotLight_Round_G_On_256c"
      ProcessValue <- "DB_HMI_sygnalizator_bocznica_krotka"
   TextField "Text field_1" at 381,92 size 71x42; Text 'pnie krótkie'
   TextField "Text field_2" at 487,91 size 72x42; Text 'pnie średnie'
   TextField "Text field_3" at 599,90 size 61x42; Text 'pnie długie'
   TextField "Text field_4" at 18,11 size 143x23; Text 'Wykryta belka:'

Template "Template_1" 800x420
   Button "Exit" at 720,360 size 78x58; TextOn 'Exit'; TextOff 'Exit'; PictureOn "ExitRuntime_TP700_Comfort_TR"; PictureOff "ExitRuntime_TP700_Comfort_TR"
      on Release: StopRuntime(0)
   Button "Template_Button" at 640,360 size 78x58; TextOff 'Text'
   Button "Template_Button_1" at 560,360 size 78x58; TextOff 'Text'
   Button "Template_Button_2" at 480,360 size 78x58; TextOff 'Text'
   Button "Template_Button_3" at 400,360 size 78x58; TextOff 'Text'
   Button "Template_Button_4" at 321,360 size 78x58; TextOff 'Text'
   Button "Template_Button_5" at 241,360 size 78x58; TextOff 'Text'
   Button "Template_Button_6" at 161,360 size 78x58; TextOff 'Text'
   Button "Template_Button_7" at 81,360 size 78x58; TextOff 'Text'
   Button "Start screen" at 1,360 size 78x58; TextOn 'Start screen'; TextOff 'Start screen'; PictureOn "NavigateHome_TP700_Comfort_TR"; PictureOff "NavigateHome_TP700_Comfort_TR"
      on Release: ActivateScreen("Root screen", 0)
*)